// TIA Portal V19 export
TYPE "LEXCHANGETRAY_typeRoller_toWorkstationDeliver"
// stored: Access Published
   STRUCT
      feedback : "LEXCHANGETRAY_typeRoller_toWorkStationRollerFeedback";
      req { S7_SetPoint := 'True'} : "LEXCHANGETRAY_typeRoller_toWorkStationRollerReq";
   END_STRUCT;
END_TYPE
